// TwinCAT 3 PLC project PlcBetterMove
// ProgramVersion: 3.1.0.8
// libraries:
//   Tc2_MC2, * (Beckhoff Automation GmbH)
//   Tc2_SerialCom, * (Beckhoff Automation GmbH)
//   Tc2_Standard, * (Beckhoff Automation GmbH)
//   Tc2_System, * (Beckhoff Automation GmbH)
//   Tc3_Interfaces, * (Beckhoff Automation GmbH)
//   Tc3_Module, * (Beckhoff Automation GmbH)
// project tree:
//   DUTs/ DATASTRUCT.TcDUT
//   GVLs/ GVL.TcGVL
//   / PlcTask.TcTTO
//   POUs/ Elbow.TcPOU, Fast.TcPOU, MAIN.TcPOU, SerialRecieve.TcPOU, WRITEFILE.TcPOU
// real-time tasks:
//   TASK PlcTask: cycle T#10ms, priority 20, ADS port 350
//   TASK CppTask: cycle T#10ms, priority 1, ADS port 351
// motion (NC):
//   TASK NC-Task 1 SAF: cycle T#2ms, priority 4, ADS port 501
//   TASK NC-Task 1 SVB: cycle T#10ms, priority 8, ADS port 511
//   AXIS Axis 1 (id 1)
//     Velo: SlowManual=2, FastManual=4, Maximum=13
//     OtherSettings: AllowMotionCmdToSlave=true
//     encoder EncType=19
//       EncPara: MaxCount=#xffffffff
//     drive DrvType=16
//       DrvPara: MaxCount=#xffffffff
//         Analog: VeloReferenz=12
//         TimeComp: TaskDelayCycles=1
//     controller CtrType=1
//       CtrPara: PriorControlFactor=1
//         Observer: BandWidth=20
//   AXIS Axis 2 (id 2)
//     Velo: SlowManual=2, FastManual=4, Maximum=13
//     OtherSettings: AllowMotionCmdToSlave=true
//     encoder EncType=19
//       EncPara: MaxCount=#xffffffff
//     drive DrvType=16
//       DrvPara: MaxCount=#xffffffff
//         Analog: VeloReferenz=12
//         TimeComp: TaskDelayCycles=1
//     controller CtrType=1
//       CtrPara: PriorControlFactor=1
//         Observer: BandWidth=20
// I/O:
//   DEVICE Device 1 (EtherCAT), AmsNetId 5.39.221.128.2.1
//     Term 1 (EK1200) [EK1200-5000 EtherCAT Power supply (2A E-Bus)]
//       Term 3 (EL2502) [EL2502 2Ch. PWM output, 24V]
//       Term 4 (EL6001) [EL6001 Interface (RS232)]
//       Term 5 (EL3002) [EL3002 2Ch. Ana. Input +/-10V]
//       Term 6 (EL4104) [EL4104 4Ch. Ana. Output 0-10V, 16bit]
//       Term 7 (EL4102) [EL4102 2Ch. Ana. Output  0-10V, 16bit]
//       Term 8 (EL3008) [EL3008 8Ch. Ana. Input +/-10V]
//       Term 9 (EL6001) [EL6001 Interface (RS232)]
//       Term 10 (EK1122) [EK1122 2 port EtherCAT junction]
//         Drive 11 (Elmo Drive) [Gold EtherCAT GCON Drive Rev:0x000103F6]
//         Drive 1 (Elmo Drive) [Gold EtherCAT GCON Drive Rev:0x000103F6]
//       Term 13 (EL6002) [EL6002 Interface 2Ch. (RS232)]
//       Term 13 (EL9011) [EL9011 End Terminal]
// variable links:
//   Device 1 (EtherCAT) <-> CppBetterMove/CppBetterMove_Obj1 (CGivePosition)
//     Term 1 (EK1200)/Term 6 (EL4104)/AO Output Channel 1/Analog output <-> Outputs/m1Int
//     Term 1 (EK1200)/Term 6 (EL4104)/AO Output Channel 2/Analog output <-> Outputs/m2Int
//   NC-Task 1 SAF/Axes/Axis 1 <-> Device 1 (EtherCAT)/Term 1 (EK1200)/Term 10 (EK1122)/Drive 11 (Elmo Drive)
//     Drive/Inputs/In/nDcOutputTime <-> InfoData/DcOutputShift
//     Drive/Inputs/In/nState1 <-> Inputs/Status word
//     Drive/Inputs/In/nState2 <-> Inputs/Status word @bit 8
//     Drive/Inputs/In/nState4 @bit 1 <-> WcState/InputToggle
//     Drive/Inputs/In/nState4 <-> WcState/WcState
//     Drive/Outputs/Out/nCtrl1 <-> Outputs/Control word
//     Drive/Outputs/Out/nCtrl2 <-> Outputs/Control word @bit 8
//     Drive/Outputs/Out/nDataOut1 <-> Outputs/Target Position
//     Enc/Inputs/In/nDataIn1 <-> Inputs/Position actual value
//     Enc/Inputs/In/nDcInputTime <-> InfoData/DcInputShift
//     Enc/Inputs/In/nState4 @bit 1 <-> WcState/InputToggle
//     Enc/Inputs/In/nState4 <-> WcState/WcState
//   NC-Task 1 SAF/Axes/Axis 2 <-> Device 1 (EtherCAT)/Term 1 (EK1200)/Term 10 (EK1122)/Drive 1 (Elmo Drive)
//     Drive/Inputs/In/nDcOutputTime <-> InfoData/DcOutputShift
//     Drive/Inputs/In/nState1 <-> Inputs/Status word
//     Drive/Inputs/In/nState2 <-> Inputs/Status word @bit 8
//     Drive/Inputs/In/nState4 @bit 1 <-> WcState/InputToggle
//     Drive/Inputs/In/nState4 <-> WcState/WcState
//     Drive/Outputs/Out/nCtrl1 <-> Outputs/Control word
//     Drive/Outputs/Out/nCtrl2 <-> Outputs/Control word @bit 8
//     Drive/Outputs/Out/nDataOut1 <-> Outputs/Target Position
//     Enc/Inputs/In/nDataIn1 <-> Inputs/Position actual value
//     Enc/Inputs/In/nDcInputTime <-> InfoData/DcInputShift
//     Enc/Inputs/In/nState4 @bit 1 <-> WcState/InputToggle
//     Enc/Inputs/In/nState4 <-> WcState/WcState
//   PlcBetterMove/PlcBetterMove Instance <-> Device 1 (EtherCAT)/Term 1 (EK1200)/Term 4 (EL6001)
//     PlcTask Inputs/GVL.EL6_22Bin_PC1/D <-> COM Inputs/Data In 0
//     PlcTask Inputs/GVL.EL6_22Bin_PC1/D @bit {8..168 step 8} <-> COM Inputs/Data In {1..21}  (21 links)
//     PlcTask Inputs/GVL.EL6_22Bin_PC1/Status <-> COM Inputs/Status
//     PlcTask Outputs/GVL.EL6_22Bout_PC1/Ctrl <-> COM Outputs/Ctrl
//     PlcTask Outputs/GVL.EL6_22Bout_PC1/D <-> COM Outputs/Data Out 0
//     PlcTask Outputs/GVL.EL6_22Bout_PC1/D @bit {8..168 step 8} <-> COM Outputs/Data Out {1..21}  (21 links)
//   PlcBetterMove/PlcBetterMove Instance <-> NC-Task 1 SAF/Axes/Axis 1
//     PlcTask Inputs/MAIN.axis1.NcToPlc <-> Outputs/ToPlc
//     PlcTask Outputs/MAIN.axis1.PlcToNc <-> Inputs/FromPlc
//   PlcBetterMove/PlcBetterMove Instance <-> CppBetterMove/CppBetterMove_Obj1 (CGivePosition)
//     PlcTask Inputs/Elbow.m1v <-> Outputs/m1v
//     PlcTask Inputs/Elbow.m2v <-> Outputs/m2v
//     PlcTask Inputs/Elbow.rad <-> Outputs/rad
//     PlcTask Inputs/Elbow.tarrad <-> Outputs/tarrad
//     PlcTask Inputs/MAIN.GivenPosition <-> Outputs/GivenPosition
//     PlcTask Inputs/MAIN.IsGivenPosition <-> Outputs/IsGivenPositon
//     PlcTask Outputs/Elbow.t <-> Inputs/PlcTimer
//     PlcTask Outputs/GVL.JIAODU <-> Inputs/Angle
//     PlcTask Outputs/MAIN.CanGivenPosition <-> Inputs/CanGivenPosition
//     PlcTask Outputs/MAIN.NextPosition <-> Inputs/NextPosition

CONFIGURATION PlcBetterMove
    RESOURCE PLC ON TwinCAT3
        TASK PlcTask(INTERVAL := T#10ms, PRIORITY := 20);
        PROGRAM Fast WITH PlcTask : Fast;
        PROGRAM Elbow WITH PlcTask : Elbow;
        PROGRAM WRITEFILE WITH PlcTask : WRITEFILE;
        PROGRAM MAIN WITH PlcTask : MAIN;
        PROGRAM SerialRecieve WITH PlcTask : SerialRecieve;
    END_RESOURCE
END_CONFIGURATION

// ---- DUTs/DATASTRUCT.TcDUT
TYPE DATASTRUCT :
STRUCT
	p1:REAL;
	p2:REAL;
	p3:REAL;
	p4:REAL;
	p5:REAL;
	g:BOOL;
	h:BOOL;
END_STRUCT
END_TYPE

// ---- GVLs/GVL.TcGVL
VAR_GLOBAL
	//读取编码器角度
	EL6_22Bin_PC1	AT %I* 	: KL6inData22b;
	EL6_22Bout_PC1	AT %Q*	: KL6outData22b;
	RxBuffer1: COMBuffer;
	TxBuffer1: COMBuffer;
	JIAODU	AT %Q* : REAL;(*单位 度*)
	JIAOSUDU: REAL;(*单位 度*)
	JIAOJIASUDU: REAL;(*单位 度*)
	//往工控机存数据
	DATA :ARRAY[1..200] OF  DATASTRUCT :=[(p1:=0,p2:=0,p2:=0,g:=FALSE,h:=FALSE)];
	bWRITE_TO_FILE:BOOL:=TRUE;
END_VAR

// ---- POUs/Fast.TcPOU
PROGRAM Fast
VAR
	SerialLineControl1:SerialLineControl;
END_VAR

//编码器任务周期
serial1fast();

ACTION Serial1Fast:
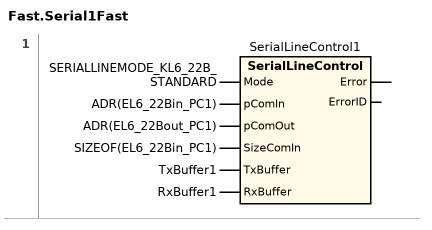
// NETWORK 1
SerialLineControl1(
    Mode := SERIALLINEMODE_KL6_22B_STANDARD,
    pComIn := ADR(EL6_22Bin_PC1),
    pComOut := ADR(EL6_22Bout_PC1),
    SizeComIn := SIZEOF(EL6_22Bin_PC1),
    TxBuffer := TxBuffer1,
    RxBuffer := RxBuffer1); // SerialLineControl
END_ACTION

END_PROGRAM

// ---- POUs/Elbow.TcPOU
PROGRAM Elbow
VAR
	t AT %Q*: REAL := 0;
	tip : REAL := 0.01;
	tarrad AT %I* : REAL;
	rad AT %I* : REAL;
	m1v AT %I* : REAL;
	m2v AT %I* : REAL;
	err: REAL;
	test AT %Q* : INT;
	a0 AT %Q* : INT;
	a1 AT %Q* : INT;
	a2 AT %Q* : INT;
	a3 AT %Q* : INT;
	a4 AT %Q* : INT;
	a5 AT %Q* : INT;
    N_save: INT := 1;
    ERRORCODE: INT := 0;
	
	v1 AT %I* : INT;
END_VAR

t := t + tip;
rad;
tarrad;
err := tarrad - rad;
m1v;
m2v;

(*IF  DATA[N_save].g=DATA[N_save].h THEN
		DATA[N_save].p1:=v1;
		DATA[N_save].g:=NOT DATA[N_save].g ;
		N_save:=N_save+1;
		IF  N_save>200 THEN
			N_save:=1;
		END_IF
ELSE
		ERRORCODE:=1;
END_IF*)


IF  DATA[N_save].g=DATA[N_save].h THEN
		DATA[N_save].p1:=tarrad;
		DATA[N_save].p2:=rad;
		DATA[N_save].p3:=err;
		DATA[N_save].p4:=m1v;
		DATA[N_save].p5:=m2v;
		DATA[N_save].g:=NOT DATA[N_save].g ;
		N_save:=N_save+1;
		IF  N_save>200 THEN
			N_save:=1;
		END_IF
ELSE
		ERRORCODE:=1;
END_IF

//IF t<6 THEN
//test := REAL_TO_INT(1*t/6.0*10000);
//a0 := REAL_TO_INT(1*t/6.0*10000);
//a1 := REAL_TO_INT(1*t/6.0*10000);
//a2 := REAL_TO_INT(1*t/6.0*10000);
//a3 := REAL_TO_INT(1*t/6.0*10000);
//a4 := REAL_TO_INT(1*t/6.0*10000);
//a5 := REAL_TO_INT(1*t/6.0*10000);
//END_IF
//IF t>6 AND t<12 THEN
//a4 := REAL_TO_INT(1*(t-6)/6.0*10000);
//END_IF
//IF t>12 AND t<18 THEN
//a1 := REAL_TO_INT(1*(18-t)/6.0*10000);
//a2 := REAL_TO_INT(1*(18-t)/6.0*10000);
//a4 := REAL_TO_INT(1*(18-t)/6.0*10000);
//END_IF

END_PROGRAM

// ---- POUs/WRITEFILE.TcPOU
PROGRAM WRITEFILE
VAR
    FILEOPEN1: FB_FileOpen;
	bFILEOPEN1: BOOL:=FALSE;
	hFile1		: UINT;
	FILEWRITE1:FB_FileWrite;
	FILECLOSE1:FB_FileClose;
	bFILECLOSE1: BOOL:=FALSE;
	bFILEWRITE1: BOOL := FALSE;
	STEP:INT:=0;
	N_SAVE:DWORD := 1;
	N_SAVE_TOTAL: DWORD := 1;
	str:STRING(200);
	N:DWORD:=1;
END_VAR

//将数值写入到工控机中
IF  bWRITE_TO_FILE THEN
	CASE STEP OF
	0:
		FILEOPEN1.bExecute:=FALSE;
		STEP:=1;
	1:
		FILEOPEN1.bExecute:=TRUE;
		FILECLOSE1.bExecute:=FALSE;
		STEP:=11;
	11:
		IF FILEOPEN1.bBusy=FALSE AND FILEOPEN1.bError=FALSE THEN
			hFile1:=FILEOPEN1.hFile;
			FILEWRITE1.bExecute:=FALSE;
			STEP:=2;
		END_IF
	2:
		IF  FILEWRITE1.bBusy=FALSE AND DATA[N_SAVE].g<>DATA[N_SAVE].h THEN
			str:=CONCAT (DWORD_TO_STRING(N_SAVE_TOTAL),' ');
			str:=CONCAT (str,REAL_TO_STRING(DATA[N_SAVE].p1));
			str:=CONCAT (str,' ');
			str:=CONCAT (str,REAL_TO_STRING(DATA[N_SAVE].p2));
			str:=CONCAT (str,' ');
			str:=CONCAT (str,REAL_TO_STRING(DATA[N_SAVE].p3));
			str:=CONCAT (str,'$n');
			FILEWRITE1.pWriteBuff:=ADR(str);
			FILEWRITE1.cbWriteLen:=LEN(str);
			FILEWRITE1.bExecute:=TRUE;
			DATA[N_SAVE].h:=NOT DATA[N_SAVE].h ;
			N_SAVE:=N_SAVE+1;
			N_SAVE_TOTAL:=N_SAVE_TOTAL+1;
			IF N_SAVE>200 THEN
			   N_SAVE:=1;
			END_IF
		END_IF;
		IF N_SAVE_TOTAL>800000 THEN
			STEP:=3;
		ELSE
			STEP:=20;
		END_IF
	20:
		FILEWRITE1.bExecute:=FALSE;
		STEP:=2;
    3:
		FILECLOSE1.bExecute:=TRUE;
		STEP:=4;
	4:
		;
	ELSE
		;
	END_CASE

END_IF

FILEOPEN1.ePath:=PATH_GENERIC;
FILEOPEN1.nMode:=FOPEN_MODEWRITE  OR FOPEN_MODETEXT ;
FILEOPEN1.sNetId:='';
FILEOPEN1.sPathName:='C:\plcwtest.txt';
FILEOPEN1.tTimeout:=t#2s;

FILEWRITE1.hFile:=hFile1;
FILEWRITE1.tTimeout:=t#1s;
FILEWRITE1.sNetId:='';

FILECLOSE1.hFile:=hFile1;
FILECLOSE1.tTimeout:=t#3s;

FILEOPEN1();
FILEWRITE1();
FILECLOSE1();

N:=N+1;

END_PROGRAM

// ---- POUs/MAIN.TcPOU
PROGRAM MAIN
VAR
	MC_Power1: MC_Power;
	MC_MoveAbsolute1: MC_MoveAbsolute;
	MC_ExtSetPointGenDisable1: MC_ExtSetPointGenDisable;
	MC_ExtSetPointGenEnable1: MC_ExtSetPointGenEnable;
	MC_Reset1: MC_Reset;
	MC_Power2: MC_Power;
	MC_MoveAbsolute2: MC_MoveAbsolute;
	axis1: AXIS_REF;				//NC轴变量
	axis2: AXIS_REF;				//NC轴变量
	status: INT;					//状态变量
//	MoveTime: LREAL := 0;			//两点间移动时间
	PlcCycleTime: LREAL := 0.01;	//PLC循环时间
	EachTime: LREAL := 2;			//距离曲线离散后,时间间隔T
	step: LREAL;					//单次移动距离
	ActGivenPosition: LREAL;		//实际给电机的坐标
	LastPosition: LREAL;			//上次实际给电机的坐标
	NextPosition AT%Q* : LREAL;			//要去的下一个给定距离
	GivenPosition AT%I* : LREAL;	//给定位置,C++输入给定位置
	CanGivenPosition AT%Q* : BOOL := FALSE;	//是否可以给定位置,输出给C++，还未做
	IsGivenPosition AT%I* : BOOL := FALSE;	//是否有给定位置,C++输入判定
	InitPosition: LREAL := 0;		//机械臂初始化位置
	
	//测试用变量
	testcount: INT;					//数组计数
	MyGivenPosition : ARRAY[0..10] OF LREAL;
	//测试用变量结束
					
END_VAR

MC_Power1(
	Axis:= axis1,
	Enable_Positive:= TRUE,
	Enable_Negative:= TRUE, );
	
MC_MoveAbsolute1(  //初始化位置
	Axis:= axis1, );
	
MC_ExtSetPointGenDisable1(
	Axis:= axis1, );
	
MC_ExtSetPointGenEnable1(
	Axis:= axis1, );
	
MC_Power2(
	Axis:= axis2,
	Enable_Positive:= TRUE,
	Enable_Negative:= TRUE, );
	
MC_MoveAbsolute2(  //初始化位置
	Axis:= axis2, );

CASE status OF
	0://init 初始化
		MC_Power1.Enable := FALSE;
		MC_ExtSetPointGenEnable1.Execute := FALSE;
		MC_ExtSetPointGenDisable1.Execute := FALSE;
		MC_MoveAbsolute1.Execute := FALSE;
		
		MC_Power2.Enable := FALSE;
		MC_MoveAbsolute2.Execute := FALSE;
		status := 1;
	1://power 使能
		MC_Power1.Enable := TRUE;
		MC_Power2.Enable := TRUE;
		IF MC_Power1.Status AND MC_Power2.Status THEN
			status := 2;
		END_IF
	2://move 移动到初始位置
		MC_MoveAbsolute1.Position := InitPosition;
		MC_MoveAbsolute1.Velocity := 2;
		MC_MoveAbsolute1.Execute := TRUE;
		MC_MoveAbsolute2.Position := 0;
		MC_MoveAbsolute2.Velocity := 1;
		MC_MoveAbsolute2.Execute := TRUE;
		IF MC_MoveAbsolute1.Done AND MC_MoveAbsolute2.Done THEN
			MC_MoveAbsolute1.Execute := FALSE;
			MC_MoveAbsolute2.Execute := FALSE;
			CanGivenPosition := TRUE;			//进入判断前一个时间,才将允许给定标志量变为真
			status := 3;
		END_IF
	3://等待变量输入,并计算单次移动距离
		IF IsGivenPosition THEN
			LastPosition := axis1.NcToPlc.ActPos;//读取当前位置作为上次给定位置
			//将一个离散时间常数内的移动距离，变换为单次plc循环的移动距离
		  	//错的 step := (GivenPositon - LastGivenPosition) * PlcCycleTime * EachTime;
			step := (GivenPosition - LastPosition) * PlcCycleTime / EachTime;
			//给定位置传送给下个位置变量
			NextPosition := GivenPosition;
			CanGivenPosition := TRUE;
			status := 4;
		END_IF
		//BREAK;
	4://按照外部给定运动，若完成当次移动后还有给定，则继续移动
		MC_ExtSetPointGenEnable1.Execute := TRUE;	//TODO：感觉可移到某个CASE里
		IF MC_ExtSetPointGenEnable1.Enabled THEN
			ActGivenPosition := LastPosition + step;//移动坐标为上次坐标加上单次移动距离
			LastPosition := ActGivenPosition;
			MC_ExtSetPointGenFeed(
				Position:= ActGivenPosition,		//给定距离
				Velocity:= 0, 						//速度和加速度可设为0，让plc自己计算
				Acceleration:= 0, 
				Direction:= 1, 
				Axis:= axis1);
		END_IF
		IF ABS(ActGivenPosition - NextPosition) <= 1E-10 THEN		//判定已经走到目标位置
			//IF判定想判定等于,但是有问题,两个认为相同的浮点数之间会有一个极小的误差存在，所以不应该判断相等
			//则判定两个的差的绝对值小于一次移动的距离的绝对值.
			//精度直接判定
			
			IF IsGivenPosition THEN			//判定还有没有给定位置，若有，则继续移动，若没有，则返回状态3等待
				step := (GivenPosition - LastPosition) * PlcCycleTime / EachTime;
				LastPosition := NextPosition;//记录上次给定位置
				NextPosition := GivenPosition;
				CanGivenPosition := TRUE;	//完成一次移动，并使用上次给定后，通知c++可以继续给定
			ELSE
				status := 3;				//返回状态3，等待位置给定
			END_IF
		ELSE
			IF IsGivenPosition THEN
				CanGivenPosition := FALSE;		//只要c++给定，就禁止再次给定
			END_IF
		END_IF
		
		
END_CASE

END_PROGRAM

// ---- POUs/SerialRecieve.TcPOU
PROGRAM SerialRecieve
VAR
	i:INT;
    AA:BYTE;
	BB:BYTE;
	RxBufferStep:INT:=0;
    AA_P:BYTE;
	BB_P:BYTE;
	JIAODU_INT:INT;
	J1: REAL:=0;
	J2: REAL:=0;
	J3: REAL:=0;
	W1:REAL:=0;
	W2:REAL:=0;
	t_tip:REAL:=0.01;
END_VAR

//读取编码器的数值
	IF RxBuffer1.Count<> 0 THEN
		FOR i:=1 TO UINT_TO_INT(RxBuffer1.Count) DO
			IF RxBufferStep=3 THEN
				BB:=RxBuffer1.Buffer[RxBuffer1.RdIdx];
				AA:=AA_P;
				RxBufferStep:=0;
			END_IF
			IF RxBufferStep=2 THEN
				AA_P:=RxBuffer1.Buffer[RxBuffer1.RdIdx];
				RxBufferStep:=3;
			END_IF
			IF RxBufferStep=1 THEN
				IF RxBuffer1.Buffer[RxBuffer1.RdIdx]=90 THEN
					RxBufferStep:=2;
				ELSE
					RxBufferStep:=0;
				END_IF
			END_IF
			IF RxBuffer1.Buffer[RxBuffer1.RdIdx]=165 THEN
				RxBufferStep:=1;
			END_IF

			RxBuffer1.RdIdx:=RxBuffer1.RdIdx+1;
			IF RxBuffer1.RdIdx>300 THEN
				RxBuffer1.RdIdx:=0;
			END_IF
		END_FOR
	RxBuffer1.Count:=0;
	END_IF

	JIAODU_INT:=UINT_TO_INT(AA*256+BB);
	JIAODU:=INT_TO_REAL(JIAODU_INT)*360.0/4096.0;
	J3:=J2;
	J2:=J1;
	J1:=JIAODU;
	JIAOSUDU:=(J1-J2)/t_tip;
	W2:=W1;
	W1:=JIAOSUDU;
	JIAOJIASUDU:=(W1-W2)/t_tip;

END_PROGRAM
